FUNCTION_BLOCK Forces1
VAR_INPUT
END_VAR
VAR_OUTPUT
END_VAR
VAR
END_VAR

END_FUNCTION_BLOCK

(* stored: Version 1.1.0.1, ProductVersion 3.1.4024.11
   POU Forces1: Id {ddc47e63-eca3-4693-bd97-1701cc096492}, SpecialFunc None *)
